// TIA Portal V15.1 export
// export: Created 2024-06-21T08:41:04.7667873Z, ExportSetting WithDefaults, DisplayName Totally Integrated Automation Portal, DisplayVersion V15.1 Update 5, DisplayName TIA Portal Openness, DisplayVersion V15.1 Update 5, DisplayName SINAMICS Startdrive Advanced, DisplayVersion V15.1, DisplayName G130, G150, S120, S150, SINAMICS MV, S210, DisplayVersion V15.1, DisplayName G110M, G120, G120C, G120D, G120P, DisplayVersion V15.1, DisplayName STEP 7 Professional, DisplayVersion V15.1 Update 5, DisplayName STEP 7 Safety, DisplayVersion V15.1, DisplayName WinCC Professional, DisplayVersion V15.1 Update 5, DisplayName SIMATIC Visualization Architect, DisplayVersion V15.1
FUNCTION_BLOCK "LAnInput6Lim"   // FB1750, FBD
TITLE = LAnInput6Lim
{ S7_Optimized_Access := 'FALSE' }
AUTHOR : VCC
FAMILY : ProcEqp
NAME : AnInput
VERSION : 1.0
// ================================================================================
// This module is used to read an analogue Input value and scale it. 
// It also gives the possibility to define 6 limits (High High High, High High, 
// High, Low, Low Low and Low Low Low level) and to create 6 alarms for these 
// limits. 
// ================================================================================
// stored: AutoNumber false, IsIECCheckEnabled false, SetENOAutomatically False, UDAEnableTagReadback false
   VAR_INPUT
      I_AnInput { ExternalAccessible := 'False'; ExternalVisible := 'False'; ExternalWritable := 'False'} : Real;   // Analogue Input Value
      I_MotorActive { ExternalAccessible := 'False'; ExternalVisible := 'False'; ExternalWritable := 'False'} : Bool;
      I_EnHHHAlarm { ExternalAccessible := 'False'; ExternalVisible := 'False'; ExternalWritable := 'False'} : Bool;   // Enable HHH Limit Alarm
      I_ResHHHAlarm { ExternalAccessible := 'False'; ExternalVisible := 'False'; ExternalWritable := 'False'} : Bool;   // Reset HHH Limit Alarm
      I_EnHHAlarm { ExternalAccessible := 'False'; ExternalVisible := 'False'; ExternalWritable := 'False'} : Bool;   // Enable HH Limit Alarm
      I_ResHHAlarm { ExternalAccessible := 'False'; ExternalVisible := 'False'; ExternalWritable := 'False'} : Bool;   // Reset HH Limit Alarm
      I_EnHAlarm { ExternalAccessible := 'False'; ExternalVisible := 'False'; ExternalWritable := 'False'} : Bool;   // Enable H Limit Alarm
      I_ResHAlarm { ExternalAccessible := 'False'; ExternalVisible := 'False'; ExternalWritable := 'False'} : Bool;   // Reset H Limit Alarm
      I_EnLAlarm { ExternalAccessible := 'False'; ExternalVisible := 'False'; ExternalWritable := 'False'} : Bool;   // Enable L Limit Alarm
      I_ResLAlarm { ExternalAccessible := 'False'; ExternalVisible := 'False'; ExternalWritable := 'False'} : Bool;   // Reset L Limit Alarm
      I_EnLLAlarm { ExternalAccessible := 'False'; ExternalVisible := 'False'; ExternalWritable := 'False'} : Bool;   // Enable LL Limit Alarm
      I_ResLLAlarm { ExternalAccessible := 'False'; ExternalVisible := 'False'; ExternalWritable := 'False'} : Bool;   // Reset LL Limit Alarm
      I_EnLLLAlarm { ExternalAccessible := 'False'; ExternalVisible := 'False'; ExternalWritable := 'False'} : Bool;   // Enable LLL Limit Alarm
      I_ResLLLAlarm { ExternalAccessible := 'False'; ExternalVisible := 'False'; ExternalWritable := 'False'} : Bool;   // Reset LLL Limit Alarm
      I_AlarmResetPB { ExternalAccessible := 'False'; ExternalVisible := 'False'; ExternalWritable := 'False'} : Bool;   // Alarm reset PB
   END_VAR
   VAR_OUTPUT
      O_HHHAlarm { ExternalAccessible := 'False'; ExternalVisible := 'False'; ExternalWritable := 'False'} : Bool;   // HHH Limit Alarm
      O_HHAlarm { ExternalAccessible := 'False'; ExternalVisible := 'False'; ExternalWritable := 'False'} : Bool;   // HH Limit Alarm
      O_HAlarm { ExternalAccessible := 'False'; ExternalVisible := 'False'; ExternalWritable := 'False'} : Bool;   // H Limit Alarm
      O_LAlarm { ExternalAccessible := 'False'; ExternalVisible := 'False'; ExternalWritable := 'False'} : Bool;   // L Limit Alarm
      O_LLAlarm { ExternalAccessible := 'False'; ExternalVisible := 'False'; ExternalWritable := 'False'} : Bool;   // LL Limit Alarm
      O_LLLAlarm { ExternalAccessible := 'False'; ExternalVisible := 'False'; ExternalWritable := 'False'} : Bool;   // LLL Limit Alarm
      O_AnInputScaled : Real;   // Analogue Input value after scaling
      O_AlarmABCondition { ExternalAccessible := 'False'; ExternalVisible := 'False'; ExternalWritable := 'False'} : Bool;   // Alarm AB condition
      O_HHHReached { ExternalAccessible := 'False'; ExternalVisible := 'False'; ExternalWritable := 'False'} : Bool;   // High High High Limit Reached
      O_HHReached { ExternalAccessible := 'False'; ExternalVisible := 'False'; ExternalWritable := 'False'} : Bool;   // High High Limit Reached
      O_HReached { ExternalAccessible := 'False'; ExternalVisible := 'False'; ExternalWritable := 'False'} : Bool;   // High Limit Reached
      O_LReached { ExternalAccessible := 'False'; ExternalVisible := 'False'; ExternalWritable := 'False'} : Bool;   // Low Limit Reached
      O_LLReached { ExternalAccessible := 'False'; ExternalVisible := 'False'; ExternalWritable := 'False'} : Bool;   // Low Low Limit Reached
      O_LLLReached { ExternalAccessible := 'False'; ExternalVisible := 'False'; ExternalWritable := 'False'} : Bool;   // Low Low Low Limit Reached
      H_IAnim { ExternalAccessible := 'False'; ExternalVisible := 'False'; ExternalWritable := 'False'} : DWord;   // HMI Animation of the icon
   END_VAR
   VAR DB_SPECIFIC
      H_In : Struct   // HMI
         AnInput_HighLimit : Real;   // From HMI : High Limit For Scaling Analogue Input
         AnInput_LowLimit : Real;   // From HMI : Low Limit For Scaling Analogue Input
         HHysteresis : Real;   // From HMI : Hysteresis value for High Limits
         LHysteresis : Real;   // From HMI : Hysteresis value for Low Limits
         HHHLimitValue : Real;   // From HMI : High High High Limit Value
         HHLimitValue : Real;   // From HMI : High High Limit Value
         HLimitValue : Real;   // From HMI : High Limit Value
         LLimitValue : Real;   // From HMI : Low Limit Value
         LLLimitValue : Real;   // From HMI : Low Low Limit Value
         LLLLimitValue : Real;   // From HMI : Low Low Low Limit Value
         TimeDelay : DInt;   // From HMI : Time delay for limits
         Forcing : Bool;   // From HMI : True if forced value must be used
         ForcedAnInput : Real;   // From HMI : Forced Analogue Input Value
      END_STRUCT;
      H_Out : Struct   // HMI
         Anim : Word;   // HMI Animation of the object
         DBnr : Int;   // HMI Animation DB number
      END_STRUCT;
   END_VAR
   VAR
      HHHLimitTimer { ExternalAccessible := 'False'; ExternalVisible := 'False'; ExternalWritable := 'False'; S7_SetPoint := 'True'} : "LTimer";   // Timer HHH Limit
      HHLimitTimer { ExternalAccessible := 'False'; ExternalVisible := 'False'; ExternalWritable := 'False'; S7_SetPoint := 'True'} : "LTimer";   // Timer HH Limit
      HLimitTimer { ExternalAccessible := 'False'; ExternalVisible := 'False'; ExternalWritable := 'False'; S7_SetPoint := 'True'} : "LTimer";   // Timer H Limit
      LLimitTimer { ExternalAccessible := 'False'; ExternalVisible := 'False'; ExternalWritable := 'False'; S7_SetPoint := 'True'} : "LTimer";   // Timer L Limit
      LLLimitTimer { ExternalAccessible := 'False'; ExternalVisible := 'False'; ExternalWritable := 'False'; S7_SetPoint := 'True'} : "LTimer";   // Timer LL Limit
      LLLLimitTimer { ExternalAccessible := 'False'; ExternalVisible := 'False'; ExternalWritable := 'False'; S7_SetPoint := 'True'} : "LTimer";   // Timer LLL Limit
   END_VAR
   VAR DB_SPECIFIC
      AnInputScaled { ExternalAccessible := 'False'; ExternalVisible := 'False'; ExternalWritable := 'False'} : Real;   // Analogue Input value after scaling
      HHHTempSR { ExternalAccessible := 'False'; ExternalVisible := 'False'; ExternalWritable := 'False'} : Bool;   // Temp variable for SET/RESET
      HHTempSR { ExternalAccessible := 'False'; ExternalVisible := 'False'; ExternalWritable := 'False'} : Bool;   // Temp variable for SET/RESET
      HTempSR { ExternalAccessible := 'False'; ExternalVisible := 'False'; ExternalWritable := 'False'} : Bool;   // Temp variable for SET/RESET
      LTempSR { ExternalAccessible := 'False'; ExternalVisible := 'False'; ExternalWritable := 'False'} : Bool;   // Temp variable for SET/RESET
      LLTempSR { ExternalAccessible := 'False'; ExternalVisible := 'False'; ExternalWritable := 'False'} : Bool;   // Temp variable for SET/RESET
      LLLTempSR { ExternalAccessible := 'False'; ExternalVisible := 'False'; ExternalWritable := 'False'} : Bool;   // Temp variable for SET/RESET
      HHHlimitHyst { ExternalAccessible := 'False'; ExternalVisible := 'False'; ExternalWritable := 'False'} : Real;   // HHH Limit with Hysteresis
      HHlimitHyst { ExternalAccessible := 'False'; ExternalVisible := 'False'; ExternalWritable := 'False'} : Real;   // HH Limit with Hysteresis
      HlimitHyst { ExternalAccessible := 'False'; ExternalVisible := 'False'; ExternalWritable := 'False'} : Real;   // H Limit with Hysteresis
      LlimitHyst { ExternalAccessible := 'False'; ExternalVisible := 'False'; ExternalWritable := 'False'} : Real;   // L Limit with Hysteresis
      LLlimitHyst { ExternalAccessible := 'False'; ExternalVisible := 'False'; ExternalWritable := 'False'} : Real;   // LL Limit with Hysteresis
      LLLlimitHyst { ExternalAccessible := 'False'; ExternalVisible := 'False'; ExternalWritable := 'False'} : Real;   // LLL Limit with Hysteresis
      HHHReached { ExternalAccessible := 'False'; ExternalVisible := 'False'; ExternalWritable := 'False'} : Bool;   // Temp variable HHH Limit Reached
      HHReached { ExternalAccessible := 'False'; ExternalVisible := 'False'; ExternalWritable := 'False'} : Bool;   // Temp variable HH Limit Reached
      HReached { ExternalAccessible := 'False'; ExternalVisible := 'False'; ExternalWritable := 'False'} : Bool;   // Temp variable H Limit Reached
      LReached { ExternalAccessible := 'False'; ExternalVisible := 'False'; ExternalWritable := 'False'} : Bool;   // Temp variable L Limit Reached
      LLReached { ExternalAccessible := 'False'; ExternalVisible := 'False'; ExternalWritable := 'False'} : Bool;   // Temp variable LL Limit Reached
      LLLReached { ExternalAccessible := 'False'; ExternalVisible := 'False'; ExternalWritable := 'False'} : Bool;   // Temp variable LLL Limit Reached
      HHHAlarmAlmCond { ExternalAccessible := 'False'; ExternalVisible := 'False'; ExternalWritable := 'False'} : Bool;   // HHHAlarm alarm condition
      HHAlarmAlmCond { ExternalAccessible := 'False'; ExternalVisible := 'False'; ExternalWritable := 'False'} : Bool;   // HHAlarm alarm condition
      HAlarmAlmCond { ExternalAccessible := 'False'; ExternalVisible := 'False'; ExternalWritable := 'False'} : Bool;   // HAlarm alarm condition
      LAlarmAlmCond { ExternalAccessible := 'False'; ExternalVisible := 'False'; ExternalWritable := 'False'} : Bool;   // LAlarm alarm condition
      LLAlarmAlmCond { ExternalAccessible := 'False'; ExternalVisible := 'False'; ExternalWritable := 'False'} : Bool;   // LLAlarm alarm condition
      LLLAlarmAlmCond { ExternalAccessible := 'False'; ExternalVisible := 'False'; ExternalWritable := 'False'} : Bool;   // LLLAlarm alarm condition
      HHHAlarm { ExternalAccessible := 'False'; ExternalVisible := 'False'; ExternalWritable := 'False'} : Bool;   // HHH Limit Alarm
      HHAlarm { ExternalAccessible := 'False'; ExternalVisible := 'False'; ExternalWritable := 'False'} : Bool;   // HH Limit Alarm
      HAlarm { ExternalAccessible := 'False'; ExternalVisible := 'False'; ExternalWritable := 'False'} : Bool;   // H Limit Alarm
      LAlarm { ExternalAccessible := 'False'; ExternalVisible := 'False'; ExternalWritable := 'False'} : Bool;   // L Limit Alarm
      LLAlarm { ExternalAccessible := 'False'; ExternalVisible := 'False'; ExternalWritable := 'False'} : Bool;   // LL Limit Alarm
      LLLAlarm { ExternalAccessible := 'False'; ExternalVisible := 'False'; ExternalWritable := 'False'} : Bool;   // LLL Limit Alarm
      AnInputTmp { ExternalAccessible := 'False'; ExternalVisible := 'False'; ExternalWritable := 'False'} : Real;   // Analog input temporary
      DBnr { ExternalAccessible := 'False'; ExternalVisible := 'False'; ExternalWritable := 'False'} : Int;   // HMI DB number
   END_VAR
   VAR
      HHH_Alarm { ExternalAccessible := 'False'; ExternalVisible := 'False'; ExternalWritable := 'False'; S7_SetPoint := 'True'} : "L1AlarmMultiIn";
      HH_Alarm { ExternalAccessible := 'False'; ExternalVisible := 'False'; ExternalWritable := 'False'; S7_SetPoint := 'True'} : "L1AlarmMultiIn";
      H_Alarm { ExternalAccessible := 'False'; ExternalVisible := 'False'; ExternalWritable := 'False'; S7_SetPoint := 'True'} : "L1AlarmMultiIn";
      L_Alarm { ExternalAccessible := 'False'; ExternalVisible := 'False'; ExternalWritable := 'False'; S7_SetPoint := 'True'} : "L1AlarmMultiIn";
      LL_Alarm { ExternalAccessible := 'False'; ExternalVisible := 'False'; ExternalWritable := 'False'; S7_SetPoint := 'True'} : "L1AlarmMultiIn";
      LLL_Alarm { ExternalAccessible := 'False'; ExternalVisible := 'False'; ExternalWritable := 'False'; S7_SetPoint := 'True'} : "L1AlarmMultiIn";
   END_VAR
BEGIN

NETWORK
TITLE = **** 1 - Inputs **** DB number
// DB number
      L     DINO;
      T     #DBnr;

REGION Network 2: **** 2.2 - Alarms - Alarm generation **** Alarm High High High Limit
   // Alarm High High High Limit
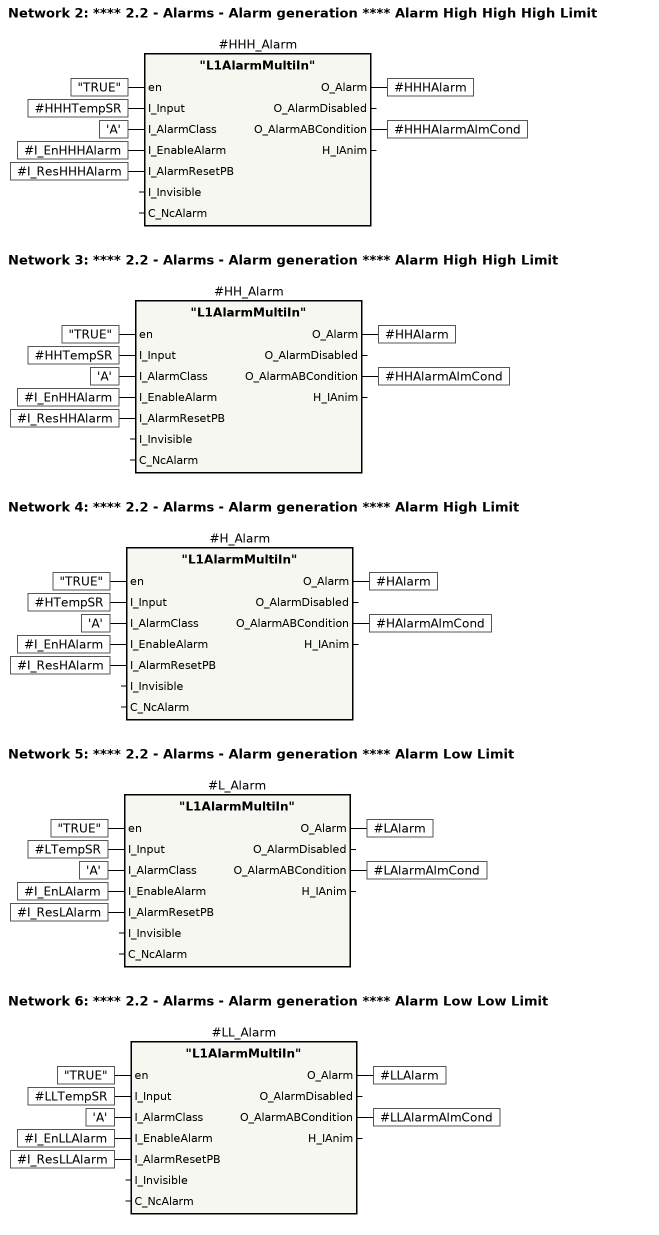
   IF "TRUE" THEN
       #HHH_Alarm(I_Input := #HHHTempSR,   // "L1AlarmMultiIn"
                  I_AlarmClass := 'A',
                  I_EnableAlarm := #I_EnHHHAlarm,
                  I_AlarmResetPB := #I_ResHHHAlarm,
                  O_Alarm => #HHHAlarm,
                  O_AlarmABCondition => #HHHAlarmAlmCond);
   END_IF;
END_REGION

REGION Network 3: **** 2.2 - Alarms - Alarm generation **** Alarm High High Limit
   // Alarm High High Limit
   IF "TRUE" THEN
       #HH_Alarm(I_Input := #HHTempSR,   // "L1AlarmMultiIn"
                 I_AlarmClass := 'A',
                 I_EnableAlarm := #I_EnHHAlarm,
                 I_AlarmResetPB := #I_ResHHAlarm,
                 O_Alarm => #HHAlarm,
                 O_AlarmABCondition => #HHAlarmAlmCond);
   END_IF;
END_REGION

REGION Network 4: **** 2.2 - Alarms - Alarm generation **** Alarm High Limit
   // Alarm High Limit
   IF "TRUE" THEN
       #H_Alarm(I_Input := #HTempSR,   // "L1AlarmMultiIn"
                I_AlarmClass := 'A',
                I_EnableAlarm := #I_EnHAlarm,
                I_AlarmResetPB := #I_ResHAlarm,
                O_Alarm => #HAlarm,
                O_AlarmABCondition => #HAlarmAlmCond);
   END_IF;
END_REGION

REGION Network 5: **** 2.2 - Alarms - Alarm generation **** Alarm Low Limit
   // Alarm Low Limit
   IF "TRUE" THEN
       #L_Alarm(I_Input := #LTempSR,   // "L1AlarmMultiIn"
                I_AlarmClass := 'A',
                I_EnableAlarm := #I_EnLAlarm,
                I_AlarmResetPB := #I_ResLAlarm,
                O_Alarm => #LAlarm,
                O_AlarmABCondition => #LAlarmAlmCond);
   END_IF;
END_REGION

REGION Network 6: **** 2.2 - Alarms - Alarm generation **** Alarm Low Low Limit
   // Alarm Low Low Limit
   IF "TRUE" THEN
       #LL_Alarm(I_Input := #LLTempSR,   // "L1AlarmMultiIn"
                 I_AlarmClass := 'A',
                 I_EnableAlarm := #I_EnLLAlarm,
                 I_AlarmResetPB := #I_ResLLAlarm,
                 O_Alarm => #LLAlarm,
                 O_AlarmABCondition => #LLAlarmAlmCond);
   END_IF;
END_REGION

REGION Network 7: **** 2.2 - Alarms - Alarm generation **** Alarm Low Low Low Limit
   // Alarm Low Low Low Limit
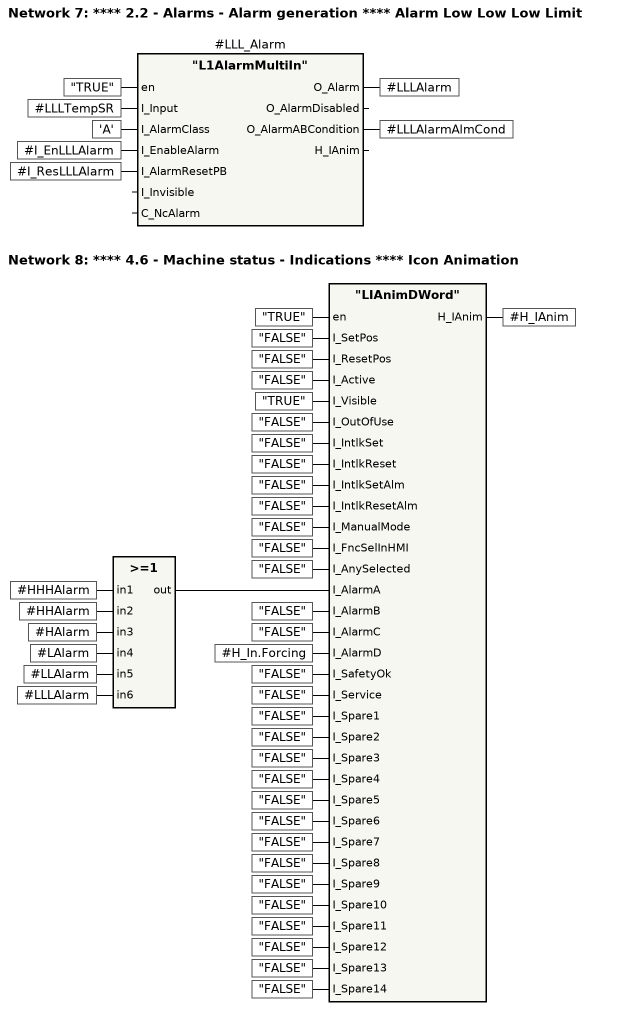
   IF "TRUE" THEN
       #LLL_Alarm(I_Input := #LLLTempSR,   // "L1AlarmMultiIn"
                  I_AlarmClass := 'A',
                  I_EnableAlarm := #I_EnLLLAlarm,
                  I_AlarmResetPB := #I_ResLLLAlarm,
                  O_Alarm => #LLLAlarm,
                  O_AlarmABCondition => #LLLAlarmAlmCond);
   END_IF;
END_REGION

REGION Network 8: **** 4.6 - Machine status - Indications **** Icon Animation
   // Icon Animation
   IF "TRUE" THEN
       "LIAnimDWord"(I_SetPos := "FALSE",
                     I_ResetPos := "FALSE",
                     I_Active := "FALSE",
                     I_Visible := "TRUE",
                     I_OutOfUse := "FALSE",
                     I_IntlkSet := "FALSE",
                     I_IntlkReset := "FALSE",
                     I_IntlkSetAlm := "FALSE",
                     I_IntlkResetAlm := "FALSE",
                     I_ManualMode := "FALSE",
                     I_FncSelInHMI := "FALSE",
                     I_AnySelected := "FALSE",
                     I_AlarmA := #HHHAlarm OR #HHAlarm OR #HAlarm OR #LAlarm OR #LLAlarm OR #LLLAlarm,
                     I_AlarmB := "FALSE",
                     I_AlarmC := "FALSE",
                     I_AlarmD := #H_In.Forcing,
                     I_SafetyOk := "FALSE",
                     I_Service := "FALSE",
                     I_Spare1 := "FALSE",
                     I_Spare2 := "FALSE",
                     I_Spare3 := "FALSE",
                     I_Spare4 := "FALSE",
                     I_Spare5 := "FALSE",
                     I_Spare6 := "FALSE",
                     I_Spare7 := "FALSE",
                     I_Spare8 := "FALSE",
                     I_Spare9 := "FALSE",
                     I_Spare10 := "FALSE",
                     I_Spare11 := "FALSE",
                     I_Spare12 := "FALSE",
                     I_Spare13 := "FALSE",
                     I_Spare14 := "FALSE",
                     H_IAnim => #H_IAnim);
   END_IF;
END_REGION

REGION Network 9: **** 4.6 - Machine status - Indications **** Animation
   // Animation
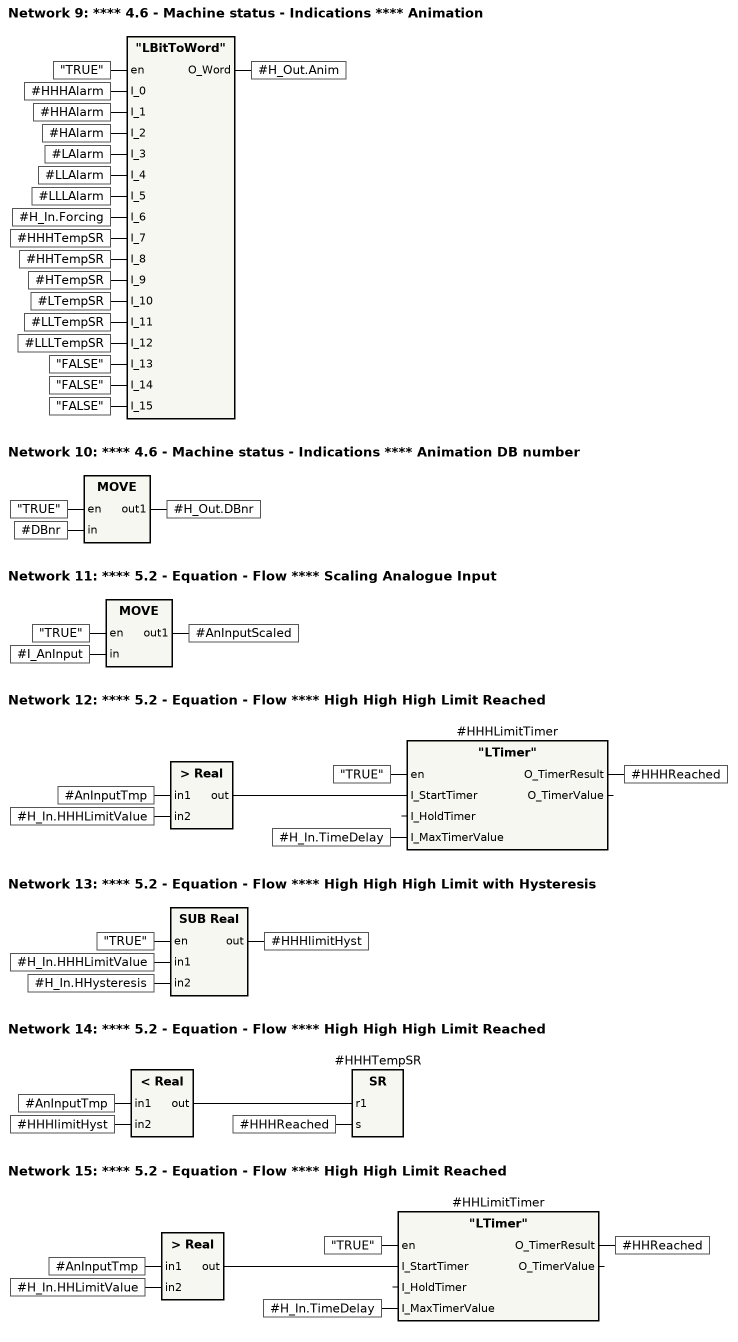
   IF "TRUE" THEN
       "LBitToWord"(I_0 := #HHHAlarm,
                    I_1 := #HHAlarm,
                    I_2 := #HAlarm,
                    I_3 := #LAlarm,
                    I_4 := #LLAlarm,
                    I_5 := #LLLAlarm,
                    I_6 := #H_In.Forcing,
                    I_7 := #HHHTempSR,
                    I_8 := #HHTempSR,
                    I_9 := #HTempSR,
                    I_10 := #LTempSR,
                    I_11 := #LLTempSR,
                    I_12 := #LLLTempSR,
                    I_13 := "FALSE",
                    I_14 := "FALSE",
                    I_15 := "FALSE",
                    O_Word => #H_Out.Anim);
   END_IF;
END_REGION

REGION Network 10: **** 4.6 - Machine status - Indications **** Animation DB number
   // Animation DB number
   IF "TRUE" THEN #H_Out.DBnr := #DBnr; END_IF;
END_REGION

REGION Network 11: **** 5.2 - Equation - Flow **** Scaling Analogue Input
   // Scaling Analogue Input
   IF "TRUE" THEN #AnInputScaled := #I_AnInput; END_IF;
END_REGION

REGION Network 12: **** 5.2 - Equation - Flow **** High High High Limit Reached
   // High High High Limit Reached
   IF "TRUE" THEN
       #HHHLimitTimer(I_StartTimer := #AnInputTmp > #H_In.HHHLimitValue,   // "LTimer"
                      I_MaxTimerValue := #H_In.TimeDelay,
                      O_TimerResult => #HHHReached);
   END_IF;
END_REGION

REGION Network 13: **** 5.2 - Equation - Flow **** High High High Limit with Hysteresis
   // High High High Limit with Hysteresis
   IF "TRUE" THEN #HHHlimitHyst := #H_In.HHHLimitValue - #H_In.HHysteresis; END_IF;
END_REGION

REGION Network 14: **** 5.2 - Equation - Flow **** High High High Limit Reached
   // High High High Limit Reached
   IF #HHHReached THEN
       #HHHTempSR := TRUE;   // SR flip-flop
   END_IF;
   IF #AnInputTmp < #HHHlimitHyst THEN #HHHTempSR := FALSE; END_IF;
END_REGION

REGION Network 15: **** 5.2 - Equation - Flow **** High High Limit Reached
   // High High Limit Reached
   IF "TRUE" THEN
       #HHLimitTimer(I_StartTimer := #AnInputTmp > #H_In.HHLimitValue,   // "LTimer"
                     I_MaxTimerValue := #H_In.TimeDelay,
                     O_TimerResult => #HHReached);
   END_IF;
END_REGION

REGION Network 16: **** 5.2 - Equation - Flow **** High High Limit with Hysteresis
   // High High Limit with Hysteresis
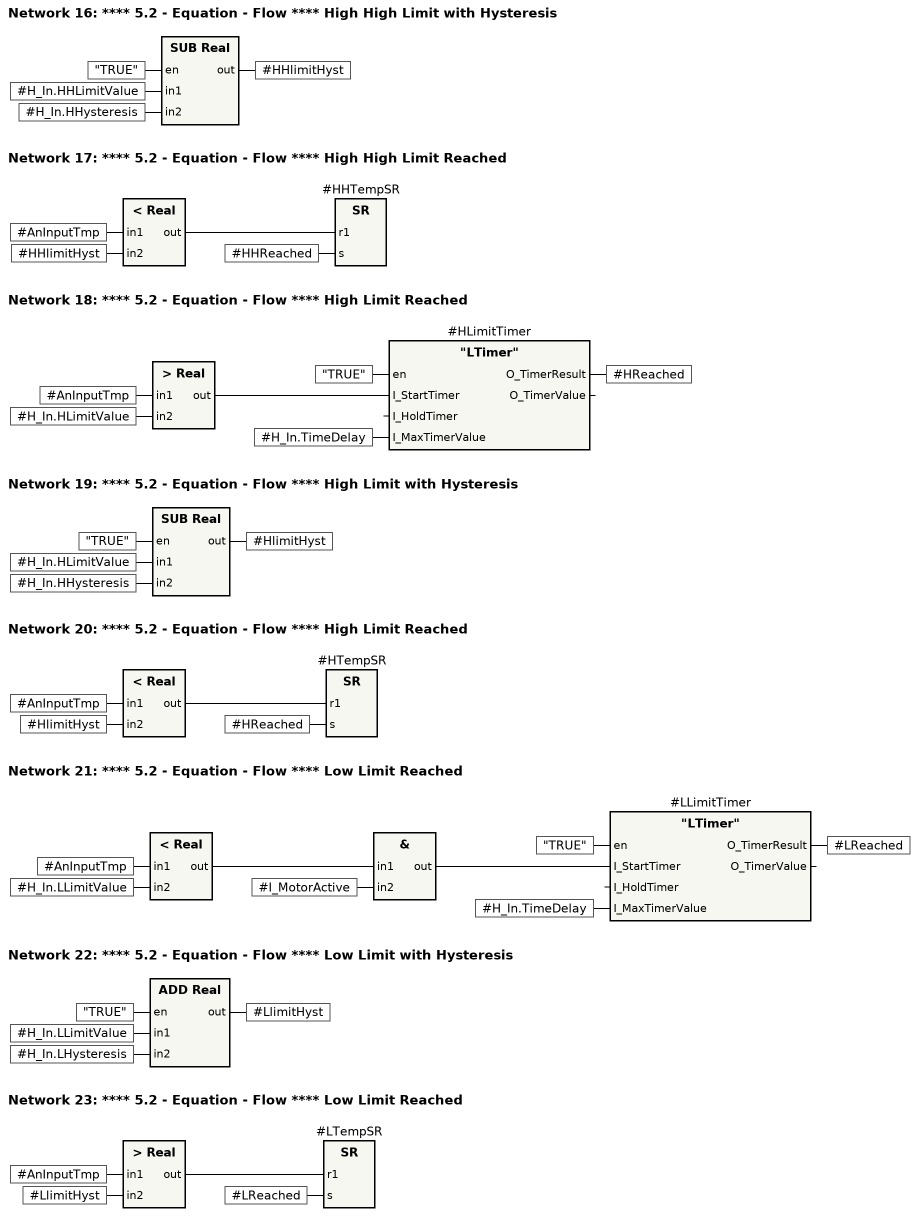
   IF "TRUE" THEN #HHlimitHyst := #H_In.HHLimitValue - #H_In.HHysteresis; END_IF;
END_REGION

REGION Network 17: **** 5.2 - Equation - Flow **** High High Limit Reached
   // High High Limit Reached
   IF #HHReached THEN
       #HHTempSR := TRUE;   // SR flip-flop
   END_IF;
   IF #AnInputTmp < #HHlimitHyst THEN #HHTempSR := FALSE; END_IF;
END_REGION

REGION Network 18: **** 5.2 - Equation - Flow **** High Limit Reached
   // High Limit Reached
   IF "TRUE" THEN
       #HLimitTimer(I_StartTimer := #AnInputTmp > #H_In.HLimitValue,   // "LTimer"
                    I_MaxTimerValue := #H_In.TimeDelay,
                    O_TimerResult => #HReached);
   END_IF;
END_REGION

REGION Network 19: **** 5.2 - Equation - Flow **** High Limit with Hysteresis
   // High Limit with Hysteresis
   IF "TRUE" THEN #HlimitHyst := #H_In.HLimitValue - #H_In.HHysteresis; END_IF;
END_REGION

REGION Network 20: **** 5.2 - Equation - Flow **** High Limit Reached
   // High Limit Reached
   IF #HReached THEN
       #HTempSR := TRUE;   // SR flip-flop
   END_IF;
   IF #AnInputTmp < #HlimitHyst THEN #HTempSR := FALSE; END_IF;
END_REGION

REGION Network 21: **** 5.2 - Equation - Flow **** Low Limit Reached
   // Low Limit Reached
   IF "TRUE" THEN
       #LLimitTimer(I_StartTimer := (#AnInputTmp < #H_In.LLimitValue) AND #I_MotorActive,   // "LTimer"
                    I_MaxTimerValue := #H_In.TimeDelay,
                    O_TimerResult => #LReached);
   END_IF;
END_REGION

REGION Network 22: **** 5.2 - Equation - Flow **** Low Limit with Hysteresis
   // Low Limit with Hysteresis
   IF "TRUE" THEN #LlimitHyst := #H_In.LLimitValue + #H_In.LHysteresis; END_IF;
END_REGION

REGION Network 23: **** 5.2 - Equation - Flow **** Low Limit Reached
   // Low Limit Reached
   IF #LReached THEN
       #LTempSR := TRUE;   // SR flip-flop
   END_IF;
   IF #AnInputTmp > #LlimitHyst THEN #LTempSR := FALSE; END_IF;
END_REGION

REGION Network 24: **** 5.2 - Equation - Flow **** Low Low Limit Reached
   // Low Low Limit Reached
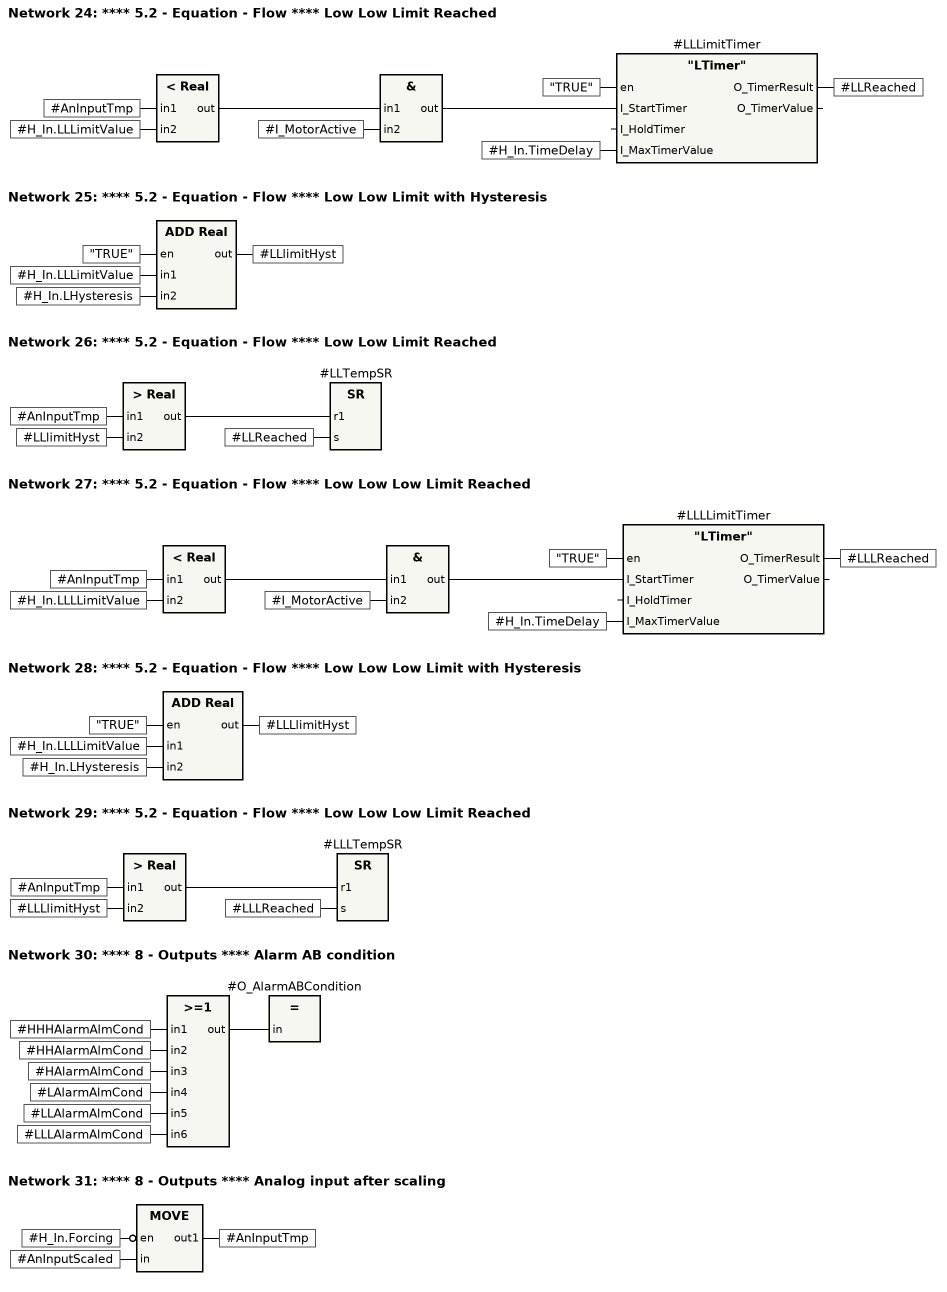
   IF "TRUE" THEN
       #LLLimitTimer(I_StartTimer := (#AnInputTmp < #H_In.LLLimitValue) AND #I_MotorActive,   // "LTimer"
                     I_MaxTimerValue := #H_In.TimeDelay,
                     O_TimerResult => #LLReached);
   END_IF;
END_REGION

REGION Network 25: **** 5.2 - Equation - Flow **** Low Low Limit with Hysteresis
   // Low Low Limit with Hysteresis
   IF "TRUE" THEN #LLlimitHyst := #H_In.LLLimitValue + #H_In.LHysteresis; END_IF;
END_REGION

REGION Network 26: **** 5.2 - Equation - Flow **** Low Low Limit Reached
   // Low Low Limit Reached
   IF #LLReached THEN
       #LLTempSR := TRUE;   // SR flip-flop
   END_IF;
   IF #AnInputTmp > #LLlimitHyst THEN #LLTempSR := FALSE; END_IF;
END_REGION

REGION Network 27: **** 5.2 - Equation - Flow **** Low Low Low Limit Reached
   // Low Low Low Limit Reached
   IF "TRUE" THEN
       #LLLLimitTimer(I_StartTimer := (#AnInputTmp < #H_In.LLLLimitValue) AND #I_MotorActive,   // "LTimer"
                      I_MaxTimerValue := #H_In.TimeDelay,
                      O_TimerResult => #LLLReached);
   END_IF;
END_REGION

REGION Network 28: **** 5.2 - Equation - Flow **** Low Low Low Limit with Hysteresis
   // Low Low Low Limit with Hysteresis
   IF "TRUE" THEN #LLLlimitHyst := #H_In.LLLLimitValue + #H_In.LHysteresis; END_IF;
END_REGION

REGION Network 29: **** 5.2 - Equation - Flow **** Low Low Low Limit Reached
   // Low Low Low Limit Reached
   IF #LLLReached THEN
       #LLLTempSR := TRUE;   // SR flip-flop
   END_IF;
   IF #AnInputTmp > #LLLlimitHyst THEN #LLLTempSR := FALSE; END_IF;
END_REGION

REGION Network 30: **** 8 - Outputs **** Alarm AB condition
   // Alarm AB condition
   #O_AlarmABCondition := #HHHAlarmAlmCond OR #HHAlarmAlmCond OR #HAlarmAlmCond OR #LAlarmAlmCond OR #LLAlarmAlmCond OR #LLLAlarmAlmCond;
END_REGION

REGION Network 31: **** 8 - Outputs **** Analog input after scaling
   // Analog input after scaling
   IF NOT #H_In.Forcing THEN #AnInputTmp := #AnInputScaled; END_IF;
END_REGION

REGION Network 32: **** 8 - Outputs **** Forcing Analogue Input
   // Forcing Analogue Input
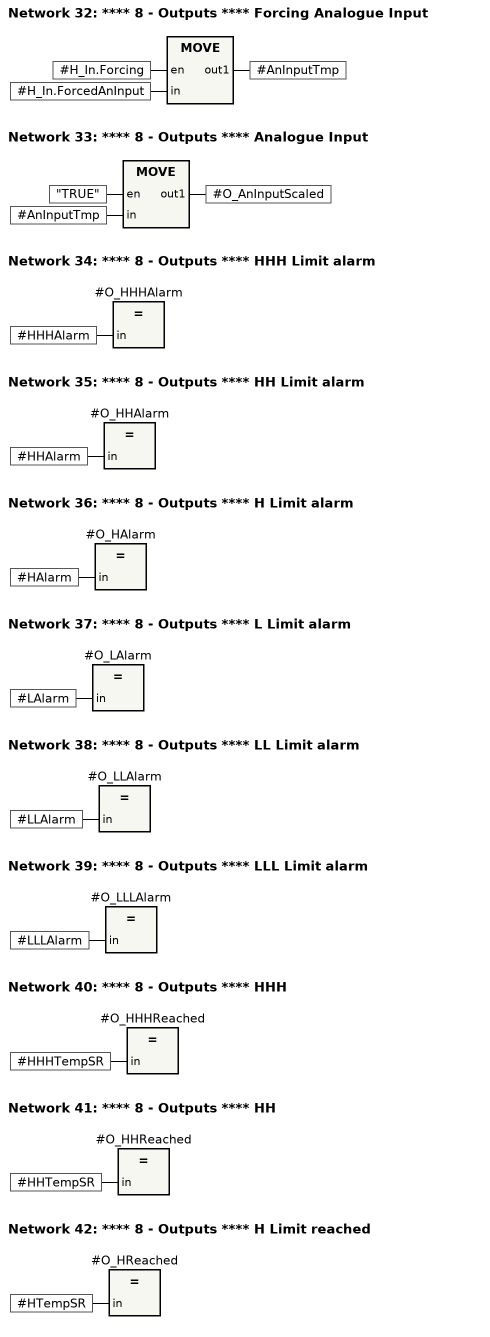
   IF #H_In.Forcing THEN #AnInputTmp := #H_In.ForcedAnInput; END_IF;
END_REGION

REGION Network 33: **** 8 - Outputs **** Analogue Input
   // Analogue Input
   IF "TRUE" THEN #O_AnInputScaled := #AnInputTmp; END_IF;
END_REGION

REGION Network 34: **** 8 - Outputs **** HHH Limit alarm
   // HHH Limit alarm
   #O_HHHAlarm := #HHHAlarm;
END_REGION

REGION Network 35: **** 8 - Outputs **** HH Limit alarm
   // HH Limit alarm
   #O_HHAlarm := #HHAlarm;
END_REGION

REGION Network 36: **** 8 - Outputs **** H Limit alarm
   // H Limit alarm
   #O_HAlarm := #HAlarm;
END_REGION

REGION Network 37: **** 8 - Outputs **** L Limit alarm
   // L Limit alarm
   #O_LAlarm := #LAlarm;
END_REGION

REGION Network 38: **** 8 - Outputs **** LL Limit alarm
   // LL Limit alarm
   #O_LLAlarm := #LLAlarm;
END_REGION

REGION Network 39: **** 8 - Outputs **** LLL Limit alarm
   // LLL Limit alarm
   #O_LLLAlarm := #LLLAlarm;
END_REGION

REGION Network 40: **** 8 - Outputs **** HHH
   // HHH
   //  Limit reached
   #O_HHHReached := #HHHTempSR;
END_REGION

REGION Network 41: **** 8 - Outputs **** HH
   // HH
   //  Limit reached
   #O_HHReached := #HHTempSR;
END_REGION

REGION Network 42: **** 8 - Outputs **** H Limit reached
   // H Limit reached
   #O_HReached := #HTempSR;
END_REGION

REGION Network 43: **** 8 - Outputs **** L Limit reached
   // L Limit reached
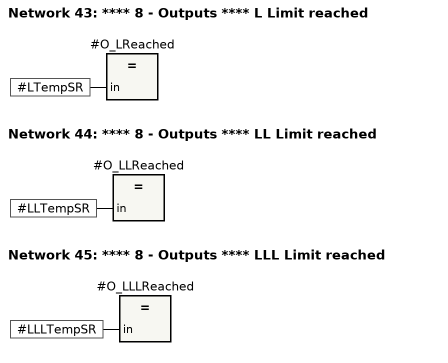
   #O_LReached := #LTempSR;
END_REGION

REGION Network 44: **** 8 - Outputs **** LL Limit reached
   // LL Limit reached
   #O_LLReached := #LLTempSR;
END_REGION

REGION Network 45: **** 8 - Outputs **** LLL Limit reached
   // LLL Limit reached
   #O_LLLReached := #LLLTempSR;
END_REGION
END_FUNCTION_BLOCK
